Universal Robots PolyScope program: Step Corner Left L.urp

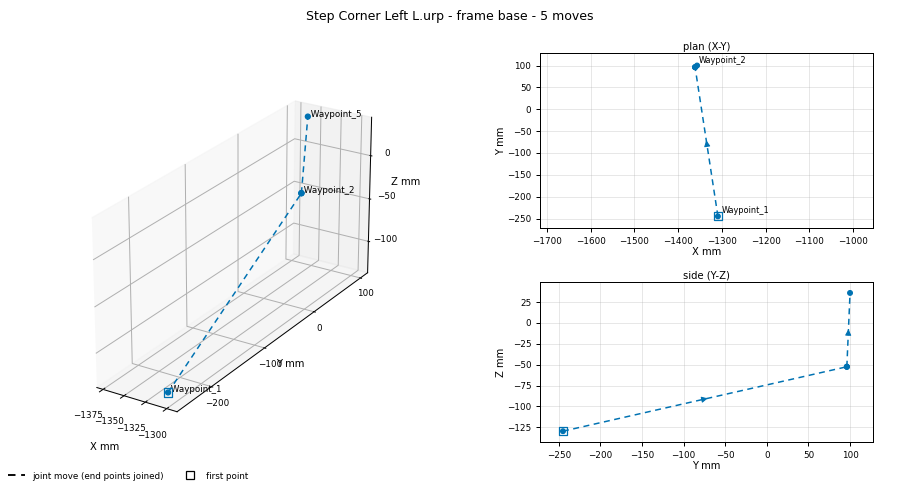
[picture p0: tool path of Step Corner Left L.urp in frame base, 5 of 5 moves have a stored position in this frame; points joined in program order, loops and branches not executed]
Program Step Corner Left L (installation=default directory=/programs createdIn=5.21.3 lastSavedIn=5.21.3 robotSerialNumber=20246801938)
Calibrated DH parameters: a=[-0.000071, -0.790281, -0.600694, 0.000061, -0.000039, 0]; d=[0.236272, 604.465945, 132.116513, -736.382239, 0.159268, 0.154005]; alpha=[1.570254, -0.000567, 0.000559, 1.571709, -1.56999, 0]; deltaTheta=[0, -0.409357, 7.293326, -0.600784, -0.000001, -0.000001]
InitVariablesNode
Robot Program (runOnlyOnce=false)
  Folder points on dummy path
    MoveJ speed 60 deg/s, acceleration 80 deg/s^2 (useActiveTCP=true optimoveEnabled=false optiMoveSpeed=0.3 optiMoveAcceleration=0.09) feature=Base
      Waypoint Waypoint_1: TCP in base x=-1309.152 y=-244.999 z=-129.703 mm, rx=-0.0526 ry=-0.0335 rz=-2.6608 rad; joints [2.155, -7.64, 72.428, -156.708, 91.75, -64.668] deg; TCP offset x=0 y=0 z=19 mm, rx=0 ry=0 rz=0 rad
      Waypoint Waypoint_2: TCP in base x=-1361.382 y=96.154 z=-52.467 mm, rx=-0.8836 ry=-1.3886 rz=-0.811 rad; joints [0.305, -9.76, 82.225, -164.326, 91.806, -62.818] deg; TCP offset x=-9.5 y=-328 z=105.73 mm, rx=1.2092 ry=-1.2092 rz=1.2092 rad
      Waypoint Waypoint_3: TCP in base x=-1361.382 y=96.154 z=-52.467 mm, rx=-0.3368 ry=-1.7393 rz=-1.3665 rad; joints [-4.241, -22.073, 102.066, -133.711, 70.536, -64.366] deg
      Waypoint Waypoint_4: TCP in base x=-1361.382 y=96.154 z=-52.467 mm, rx=0.4125 ry=-1.9596 rz=-1.9004 rad; joints [-7.381, -37.593, 106.062, -73.091, 55.284, -86.525] deg
      Waypoint Waypoint_5: TCP in base x=-1356.834 y=99.984 z=35.986 mm, rx=0.4125 ry=-1.9596 rz=-1.9004 rad; joints [-7.639, -43.359, 107.418, -68.7, 55.029, -86.493] deg
